# EPICS substitutions: motorThorLabsAptApp/Db/user.substitutions
# Example substitutions file

file db/thorLabsApt.db {
    pattern { P, R, PORT, ADDR, TIMEOUT, LSCALE, VSCALE, ASCALE, UNIT }
        { "KBD101", "{DDSM100-1}", "KBD", 0, 0, 10, 10, 10, "mm" }
#        { "KBD101", "{DDSM100-2}", "KBD", 0, 0, 10, 10, 10, "mm" }
#        { "KBD101", "{DDSM100-3}", "KBD", 0, 0, 10, 10, 10, "mm" }
}
